FUNCTION WRITE_ANY_USINT : BOOL
VAR_INPUT
    ptr: POINTER TO USINT;
    val: USINT;
END_VAR

ptr^ := val;

END_FUNCTION

(* stored: Version 1.1.0.1, ProductVersion 3.1.4022.9
   POU WRITE_ANY_USINT: Id {333ffbf6-74a7-432c-9a43-c67b08c23471}, SpecialFunc None *)
